Universal Robots PolyScope program: Lab_exe_12_2_221.urp

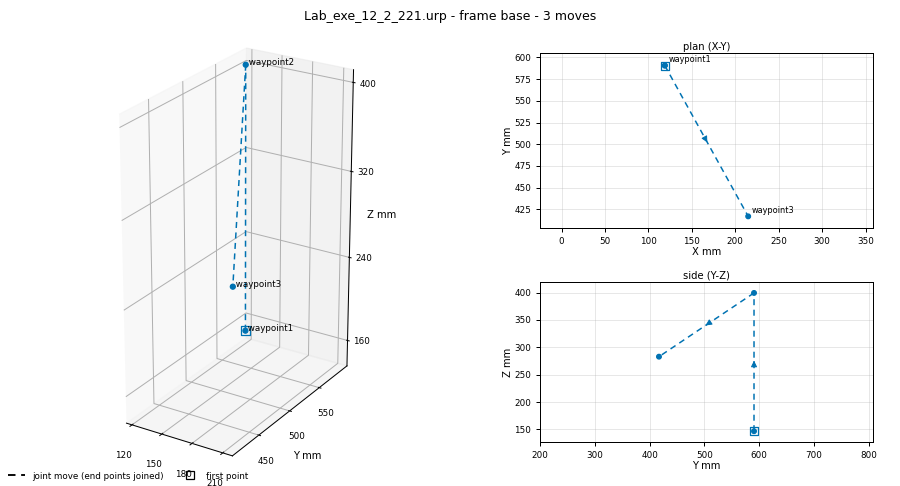
[picture p0: tool path of Lab_exe_12_2_221.urp in frame base, 3 of 3 moves have a stored position in this frame; points joined in program order, loops and branches not executed]
Program Lab_exe_12_2_221 (createdIn=3.2.19293 lastSavedIn=3.2.19293 directory=/programs installation=default robotSerialNumber=2015351391)
Calibrated DH parameters: a=[0.000352, -0.161198, -0.373486, 0.00005, 0.000049, 0]; d=[0.089268, 352.477598, -320.08558, -32.281492, 0.094939, 0.082518]; alpha=[1.570728, 0.001116, -0.003686, 1.571189, -1.570572, 0]; deltaTheta=[-0.000012, 1.181849, -1.491165, 0.309495, -0.000007, 0.000025]
Robot Program (runOnlyOnce=false motionType=MoveJ speed=1.047198 acceleration=1.396263 recalculateMotions=false)
  MoveJ speed 60 deg/s, acceleration 80 deg/s^2 (recalculateMotions=false)
    Waypoint waypoint1: TCP in base x=118.887 y=590.552 z=146.827 mm, rx=-1.1701 ry=2.6606 rz=0.3786 rad; joints [91.175, -102.305, -106.896, -42.449, 84.482, 132.6] deg; flange x=107.884 y=551.156 z=264.943 mm, rx=-1.1702 ry=2.6606 rz=0.3787 rad
    Waypoint waypoint2: TCP in base x=118.862 y=590.578 z=399.347 mm, rx=-1.1701 ry=2.6606 rz=0.3787 rad; joints [91.18, -95.976, -76.122, -79.561, 84.377, 132.702] deg; flange x=107.884 y=551.156 z=517.465 mm, rx=-1.1702 ry=2.6606 rz=0.3787 rad
    Waypoint waypoint3: TCP in base x=214.827 y=416.984 z=282.935 mm, rx=-1.1703 ry=2.6606 rz=0.3787 rad; joints [76.813, -77.666, -110.566, -62.7, 89.035, 119.044] deg; flange x=203.875 y=377.556 z=401.074 mm, rx=-1.1702 ry=2.6606 rz=0.3787 rad
